(* PLC project safeApp1, BrAutomation SafeDESIGNER  5.17.0.0 *)
(* stored: companyURL http://www.br-automation.com, creationDateTime Thu May 19 09:53:23 2022 *)

PROGRAM Main

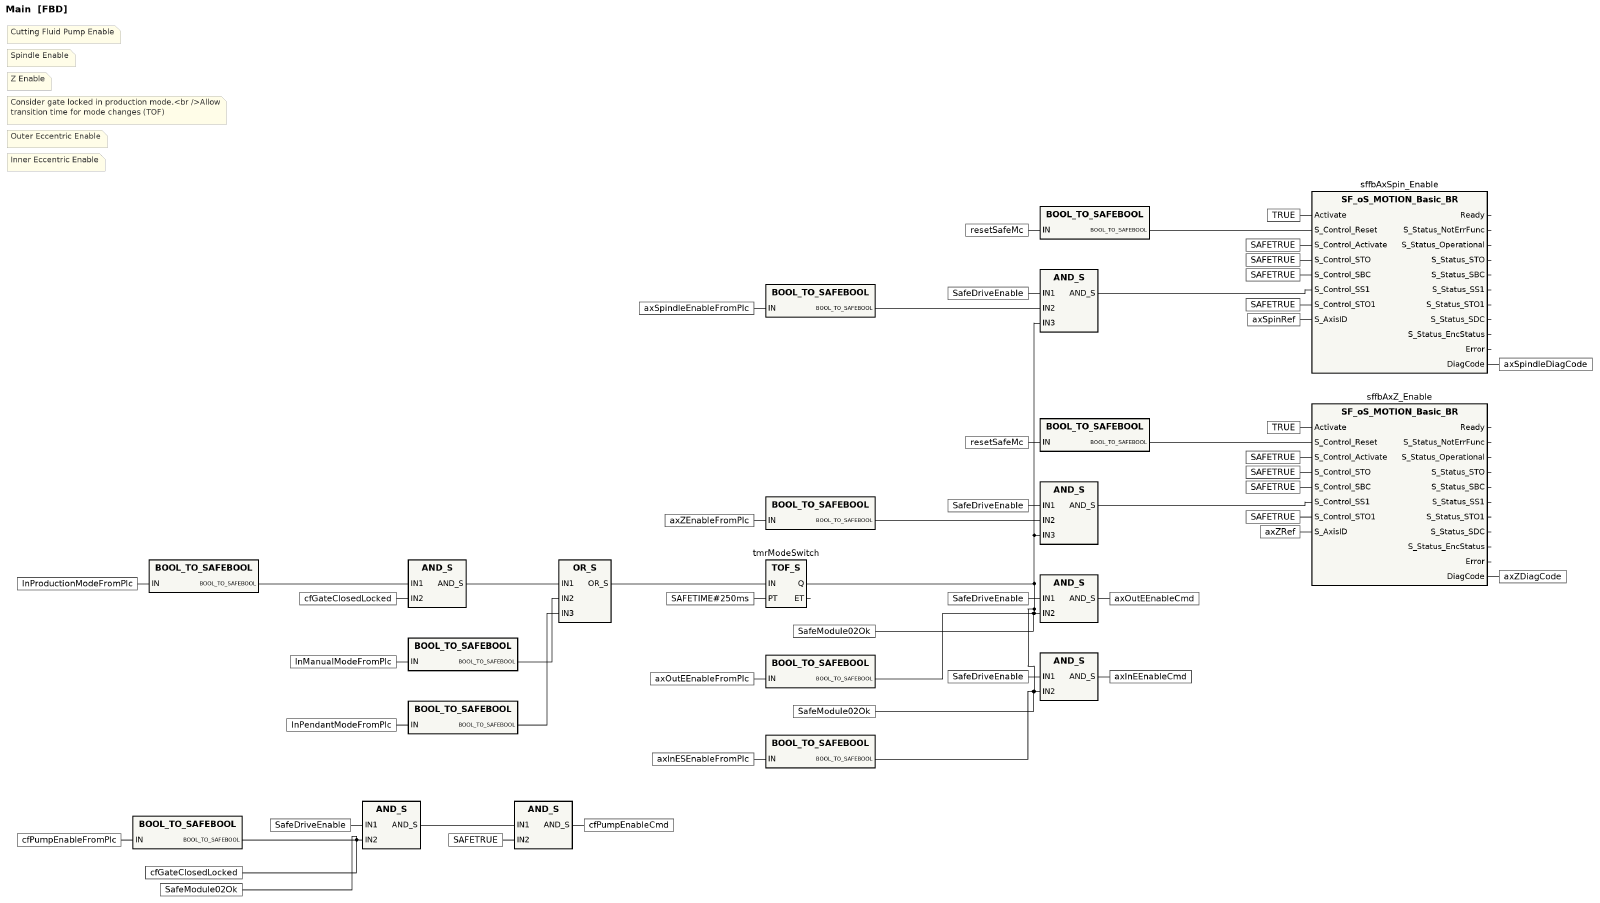
(* FBD diagram, written out as Structured Text *)
(* Spindle Enable *)
(* Consider gate locked in production mode.<br />Allow transition time for mode changes (TOF) *)
tmrModeSwitch(IN := OR_S(AND_S(BOOL_TO_SAFEBOOL(InProductionModeFromPlc), cfGateClosedLocked), BOOL_TO_SAFEBOOL(InManualModeFromPlc), BOOL_TO_SAFEBOOL(InPendantModeFromPlc)), PT := SAFETIME#250ms);
sffbAxSpin_Enable(Activate := TRUE, S_Control_Reset := BOOL_TO_SAFEBOOL(resetSafeMc), S_Control_Activate := SAFETRUE, S_Control_STO := SAFETRUE, S_Control_SBC := SAFETRUE, S_Control_SS1 := AND_S(SafeDriveEnable, BOOL_TO_SAFEBOOL(axSpindleEnableFromPlc), tmrModeSwitch.Q), S_Control_STO1 := SAFETRUE, S_AxisID := axSpinRef);
axSpindleDiagCode := sffbAxSpin_Enable.DiagCode;
(* Z Enable *)
sffbAxZ_Enable(Activate := TRUE, S_Control_Reset := BOOL_TO_SAFEBOOL(resetSafeMc), S_Control_Activate := SAFETRUE, S_Control_STO := SAFETRUE, S_Control_SBC := SAFETRUE, S_Control_SS1 := AND_S(SafeDriveEnable, BOOL_TO_SAFEBOOL(axZEnableFromPlc), tmrModeSwitch.Q), S_Control_STO1 := SAFETRUE, S_AxisID := axZRef);
axZDiagCode := sffbAxZ_Enable.DiagCode;
(* Outer Eccentric Enable *)
axOutEEnableCmd := AND_S(SafeDriveEnable, BOOL_TO_SAFEBOOL(axOutEEnableFromPlc), tmrModeSwitch.Q, SafeModule02Ok);
(* Inner Eccentric Enable *)
axInEEnableCmd := AND_S(SafeDriveEnable, BOOL_TO_SAFEBOOL(axInESEnableFromPlc), tmrModeSwitch.Q, SafeModule02Ok);
(* Cutting Fluid Pump Enable *)
cfPumpEnableCmd := AND_S(AND_S(SafeDriveEnable, BOOL_TO_SAFEBOOL(cfPumpEnableFromPlc), cfGateClosedLocked, SafeModule02Ok), SAFETRUE);
END_PROGRAM
